# EPICS substitutions: mpgSupport/Db/bsaEdefMaskUnit/bsaEdefMaskUnitAll.substitutions
#==============================================================================
#
# Abs:  Beam Synchronous Acquisition masks
#
# Name: bsaEdefMaskUnitAll.substitutions
#
# Note: Must follow the LCLS naming conventions.
#
#==============================================================================
#
file bsaEdefMaskUnit.db
{
  pattern {     MD,  MASK, INDEX,     SYS ,     DEV   }
	  { $(S_MD), INCM,   1  , $(S_SYS), $(S_DEV)  }
	  { $(S_MD), INCM,   2  , $(S_SYS), $(S_DEV)  }
	  { $(S_MD), INCM,   3  , $(S_SYS), $(S_DEV)  }
          { $(S_MD), INCM,   4  , $(S_SYS), $(S_DEV)  }
          { $(S_MD), INCM,   5  , $(S_SYS), $(S_DEV)  }
          { $(S_MD), INCM,   6  , $(S_SYS), $(S_DEV)  }
          { $(S_MD), INCM,   7  , $(S_SYS), $(S_DEV)  }
          { $(S_MD), INCM,   8  , $(S_SYS), $(S_DEV)  }
          { $(S_MD), INCM,   9  , $(S_SYS), $(S_DEV)  }
          { $(S_MD), INCM,  10  , $(S_SYS), $(S_DEV)  }
          { $(S_MD), INCM,  11  , $(S_SYS), $(S_DEV)  }
          { $(S_MD), INCM,  12  , $(S_SYS), $(S_DEV)  }
          { $(S_MD), INCM,  13  , $(S_SYS), $(S_DEV)  }
          { $(S_MD), INCM,  14  , $(S_SYS), $(S_DEV)  }
          { $(S_MD), INCM,  15  , $(S_SYS), $(S_DEV)  }
          { $(S_MD), INCM,  16  , $(S_SYS), $(S_DEV)  }
          { $(S_MD), INCM,  17  , $(S_SYS), $(S_DEV)  }
          { $(S_MD), INCM,  18  , $(S_SYS), $(S_DEV)  }
          { $(S_MD), INCM,  19  , $(S_SYS), $(S_DEV)  }
          { $(S_MD), INCM,  20  , $(S_SYS), $(S_DEV)  }
          { $(S_MD), INCM,  21  , $(S_SYS), $(S_DEV)  }
          { $(S_MD), INCM,  22  , $(S_SYS), $(S_DEV)  }
          { $(S_MD), INCM,  23  , $(S_SYS), $(S_DEV)  }
          { $(S_MD), INCM,  24  , $(S_SYS), $(S_DEV)  }
          { $(S_MD), INCM,  25  , $(S_SYS), $(S_DEV)  }
          { $(S_MD), INCM,  26  , $(S_SYS), $(S_DEV)  }
          { $(S_MD), INCM,  27  , $(S_SYS), $(S_DEV)  }
          { $(S_MD), INCM,  28  , $(S_SYS), $(S_DEV)  }
          { $(S_MD), INCM,  29  , $(S_SYS), $(S_DEV)  }
          { $(S_MD), INCM,  30  , $(S_SYS), $(S_DEV)  }
          { $(S_MD), INCM,  31  , $(S_SYS), $(S_DEV)  }
          { $(S_MD), INCM,  32  , $(S_SYS), $(S_DEV)  }
          { $(S_MD), INCM,  33  , $(S_SYS), $(S_DEV)  }
          { $(S_MD), INCM,  34  , $(S_SYS), $(S_DEV)  }
          { $(S_MD), INCM,  35  , $(S_SYS), $(S_DEV)  }
          { $(S_MD), INCM,  36  , $(S_SYS), $(S_DEV)  }
          { $(S_MD), INCM,  37  , $(S_SYS), $(S_DEV)  }
          { $(S_MD), INCM,  38  , $(S_SYS), $(S_DEV)  }
          { $(S_MD), INCM,  39  , $(S_SYS), $(S_DEV)  }
          { $(S_MD), INCM,  40  , $(S_SYS), $(S_DEV)  }
          { $(S_MD), INCM,  41  , $(S_SYS), $(S_DEV)  }
          { $(S_MD), INCM,  42  , $(S_SYS), $(S_DEV)  }
          { $(S_MD), INCM,  43  , $(S_SYS), $(S_DEV)  }
          { $(S_MD), INCM,  44  , $(S_SYS), $(S_DEV)  }
          { $(S_MD), INCM,  45  , $(S_SYS), $(S_DEV)  }
          { $(S_MD), INCM,  46  , $(S_SYS), $(S_DEV)  }
          { $(S_MD), INCM,  47  , $(S_SYS), $(S_DEV)  }
          { $(S_MD), INCM,  48  , $(S_SYS), $(S_DEV)  }
          { $(S_MD), INCM,  49  , $(S_SYS), $(S_DEV)  }
          { $(S_MD), INCM,  50  , $(S_SYS), $(S_DEV)  }
          { $(S_MD), INCM,  51  , $(S_SYS), $(S_DEV)  }
          { $(S_MD), INCM,  52  , $(S_SYS), $(S_DEV)  }
          { $(S_MD), INCM,  53  , $(S_SYS), $(S_DEV)  }
          { $(S_MD), INCM,  54  , $(S_SYS), $(S_DEV)  }
          { $(S_MD), INCM,  55  , $(S_SYS), $(S_DEV)  }
          { $(S_MD), INCM,  56  , $(S_SYS), $(S_DEV)  }
          { $(S_MD), INCM,  57  , $(S_SYS), $(S_DEV)  }
          { $(S_MD), INCM,  58  , $(S_SYS), $(S_DEV)  }
          { $(S_MD), INCM,  59  , $(S_SYS), $(S_DEV)  }
          { $(S_MD), INCM,  60  , $(S_SYS), $(S_DEV)  }
          { $(S_MD), INCM,  61  , $(S_SYS), $(S_DEV)  }
          { $(S_MD), INCM,  62  , $(S_SYS), $(S_DEV)  }
          { $(S_MD), INCM,  63  , $(S_SYS), $(S_DEV)  }
          { $(S_MD), INCM,  64  , $(S_SYS), $(S_DEV)  }
          { $(S_MD), INCM,  65  , $(S_SYS), $(S_DEV)  }
          { $(S_MD), INCM,  66  , $(S_SYS), $(S_DEV)  }
          { $(S_MD), INCM,  67  , $(S_SYS), $(S_DEV)  }
          { $(S_MD), INCM,  68  , $(S_SYS), $(S_DEV)  }
          { $(S_MD), INCM,  69  , $(S_SYS), $(S_DEV)  }
          { $(S_MD), INCM,  70  , $(S_SYS), $(S_DEV)  }
          { $(S_MD), INCM,  71  , $(S_SYS), $(S_DEV)  }
          { $(S_MD), INCM,  72  , $(S_SYS), $(S_DEV)  }
          { $(S_MD), INCM,  73  , $(S_SYS), $(S_DEV)  }
          { $(S_MD), INCM,  74  , $(S_SYS), $(S_DEV)  }
          { $(S_MD), INCM,  75  , $(S_SYS), $(S_DEV)  }
          { $(S_MD), INCM,  76  , $(S_SYS), $(S_DEV)  }
          { $(S_MD), INCM,  77  , $(S_SYS), $(S_DEV)  }
          { $(S_MD), INCM,  78  , $(S_SYS), $(S_DEV)  }
          { $(S_MD), INCM,  79  , $(S_SYS), $(S_DEV)  }
          { $(S_MD), INCM,  80  , $(S_SYS), $(S_DEV)  }
          { $(S_MD), INCM,  81  , $(S_SYS), $(S_DEV)  }
          { $(S_MD), INCM,  82  , $(S_SYS), $(S_DEV)  }
          { $(S_MD), INCM,  83  , $(S_SYS), $(S_DEV)  }
          { $(S_MD), INCM,  84  , $(S_SYS), $(S_DEV)  }
          { $(S_MD), INCM,  85  , $(S_SYS), $(S_DEV)  }
          { $(S_MD), INCM,  86  , $(S_SYS), $(S_DEV)  }
          { $(S_MD), INCM,  87  , $(S_SYS), $(S_DEV)  }
          { $(S_MD), INCM,  88  , $(S_SYS), $(S_DEV)  }
          { $(S_MD), INCM,  89  , $(S_SYS), $(S_DEV)  }
          { $(S_MD), INCM,  90  , $(S_SYS), $(S_DEV)  }
          { $(S_MD), INCM,  91  , $(S_SYS), $(S_DEV)  }
          { $(S_MD), INCM,  92  , $(S_SYS), $(S_DEV)  }
          { $(S_MD), INCM,  93  , $(S_SYS), $(S_DEV)  }
          { $(S_MD), INCM,  94  , $(S_SYS), $(S_DEV)  }
          { $(S_MD), INCM,  95  , $(S_SYS), $(S_DEV)  }
          { $(S_MD), INCM,  96  , $(S_SYS), $(S_DEV)  }
          { $(S_MD), INCM,  97  , $(S_SYS), $(S_DEV)  }
          { $(S_MD), INCM,  98  , $(S_SYS), $(S_DEV)  }
          { $(S_MD), INCM,  99  , $(S_SYS), $(S_DEV)  }
          { $(S_MD), INCM, 100  , $(S_SYS), $(S_DEV)  }
          { $(S_MD), INCM, 101  , $(S_SYS), $(S_DEV)  }
          { $(S_MD), INCM, 102  , $(S_SYS), $(S_DEV)  }
          { $(S_MD), INCM, 103  , $(S_SYS), $(S_DEV)  }
          { $(S_MD), INCM, 104  , $(S_SYS), $(S_DEV)  }
          { $(S_MD), INCM, 105  , $(S_SYS), $(S_DEV)  }
          { $(S_MD), INCM, 106  , $(S_SYS), $(S_DEV)  }
          { $(S_MD), INCM, 107  , $(S_SYS), $(S_DEV)  }
          { $(S_MD), INCM, 108  , $(S_SYS), $(S_DEV)  }
          { $(S_MD), INCM, 109  , $(S_SYS), $(S_DEV)  }
          { $(S_MD), INCM, 110  , $(S_SYS), $(S_DEV)  }
          { $(S_MD), INCM, 111  , $(S_SYS), $(S_DEV)  }
          { $(S_MD), INCM, 112  , $(S_SYS), $(S_DEV)  }
          { $(S_MD), INCM, 113  , $(S_SYS), $(S_DEV)  }
          { $(S_MD), INCM, 114  , $(S_SYS), $(S_DEV)  }
          { $(S_MD), INCM, 115  , $(S_SYS), $(S_DEV)  }
          { $(S_MD), INCM, 116  , $(S_SYS), $(S_DEV)  }
          { $(S_MD), INCM, 117  , $(S_SYS), $(S_DEV)  }
          { $(S_MD), INCM, 118  , $(S_SYS), $(S_DEV)  }
          { $(S_MD), INCM, 119  , $(S_SYS), $(S_DEV)  }
          { $(S_MD), INCM, 120  , $(S_SYS), $(S_DEV)  }
          { $(S_MD), INCM, 121  , $(S_SYS), $(S_DEV)  }
          { $(S_MD), INCM, 122  , $(S_SYS), $(S_DEV)  }
          { $(S_MD), INCM, 123  , $(S_SYS), $(S_DEV)  }
          { $(S_MD), INCM, 124  , $(S_SYS), $(S_DEV)  }
          { $(S_MD), INCM, 125  , $(S_SYS), $(S_DEV)  }
          { $(S_MD), INCM, 126  , $(S_SYS), $(S_DEV)  }
          { $(S_MD), INCM, 127  , $(S_SYS), $(S_DEV)  }
          { $(S_MD), INCM, 128  , $(S_SYS), $(S_DEV)  }
          { $(S_MD), INCM, 129  , $(S_SYS), $(S_DEV)  }
          { $(S_MD), INCM, 130  , $(S_SYS), $(S_DEV)  }
          { $(S_MD), INCM, 131  , $(S_SYS), $(S_DEV)  }
          { $(S_MD), INCM, 132  , $(S_SYS), $(S_DEV)  }
          { $(S_MD), INCM, 133  , $(S_SYS), $(S_DEV)  }
          { $(S_MD), INCM, 134  , $(S_SYS), $(S_DEV)  }
          { $(S_MD), INCM, 135  , $(S_SYS), $(S_DEV)  }
          { $(S_MD), INCM, 136  , $(S_SYS), $(S_DEV)  }
          { $(S_MD), INCM, 137  , $(S_SYS), $(S_DEV)  }
          { $(S_MD), INCM, 138  , $(S_SYS), $(S_DEV)  }
          { $(S_MD), INCM, 139  , $(S_SYS), $(S_DEV)  }
          { $(S_MD), INCM, 140  , $(S_SYS), $(S_DEV)  }
          { $(S_MD), INCM, 141  , $(S_SYS), $(S_DEV)  }
          { $(S_MD), INCM, 142  , $(S_SYS), $(S_DEV)  }
          { $(S_MD), INCM, 143  , $(S_SYS), $(S_DEV)  }
          { $(S_MD), INCM, 144  , $(S_SYS), $(S_DEV)  }
          { $(S_MD), INCM, 145  , $(S_SYS), $(S_DEV)  }
          { $(S_MD), INCM, 146  , $(S_SYS), $(S_DEV)  }
          { $(S_MD), INCM, 147  , $(S_SYS), $(S_DEV)  }
          { $(S_MD), INCM, 148  , $(S_SYS), $(S_DEV)  }
          { $(S_MD), INCM, 149  , $(S_SYS), $(S_DEV)  }
          { $(S_MD), INCM, 150  , $(S_SYS), $(S_DEV)  }
          { $(S_MD), INCM, 151  , $(S_SYS), $(S_DEV)  }
          { $(S_MD), INCM, 152  , $(S_SYS), $(S_DEV)  }
          { $(S_MD), INCM, 153  , $(S_SYS), $(S_DEV)  }
          { $(S_MD), INCM, 154  , $(S_SYS), $(S_DEV)  }
          { $(S_MD), INCM, 155  , $(S_SYS), $(S_DEV)  }
          { $(S_MD), INCM, 156  , $(S_SYS), $(S_DEV)  }
          { $(S_MD), INCM, 157  , $(S_SYS), $(S_DEV)  }
          { $(S_MD), INCM, 158  , $(S_SYS), $(S_DEV)  }
          { $(S_MD), INCM, 159  , $(S_SYS), $(S_DEV)  }
          { $(S_MD), INCM, 160  , $(S_SYS), $(S_DEV)  }

	  { $(S_MD), EXCM,   1  , $(S_SYS), $(S_DEV)  }
	  { $(S_MD), EXCM,   2  , $(S_SYS), $(S_DEV)  }
	  { $(S_MD), EXCM,   3  , $(S_SYS), $(S_DEV)  }
          { $(S_MD), EXCM,   4  , $(S_SYS), $(S_DEV)  }
          { $(S_MD), EXCM,   5  , $(S_SYS), $(S_DEV)  }
          { $(S_MD), EXCM,   6  , $(S_SYS), $(S_DEV)  }
          { $(S_MD), EXCM,   7  , $(S_SYS), $(S_DEV)  }
          { $(S_MD), EXCM,   8  , $(S_SYS), $(S_DEV)  }
          { $(S_MD), EXCM,   9  , $(S_SYS), $(S_DEV)  }
          { $(S_MD), EXCM,  10  , $(S_SYS), $(S_DEV)  }
          { $(S_MD), EXCM,  11  , $(S_SYS), $(S_DEV)  }
          { $(S_MD), EXCM,  12  , $(S_SYS), $(S_DEV)  }
          { $(S_MD), EXCM,  13  , $(S_SYS), $(S_DEV)  }
          { $(S_MD), EXCM,  14  , $(S_SYS), $(S_DEV)  }
          { $(S_MD), EXCM,  15  , $(S_SYS), $(S_DEV)  }
          { $(S_MD), EXCM,  16  , $(S_SYS), $(S_DEV)  }
          { $(S_MD), EXCM,  17  , $(S_SYS), $(S_DEV)  }
          { $(S_MD), EXCM,  18  , $(S_SYS), $(S_DEV)  }
          { $(S_MD), EXCM,  19  , $(S_SYS), $(S_DEV)  }
          { $(S_MD), EXCM,  20  , $(S_SYS), $(S_DEV)  }
          { $(S_MD), EXCM,  21  , $(S_SYS), $(S_DEV)  }
          { $(S_MD), EXCM,  22  , $(S_SYS), $(S_DEV)  }
          { $(S_MD), EXCM,  23  , $(S_SYS), $(S_DEV)  }
          { $(S_MD), EXCM,  24  , $(S_SYS), $(S_DEV)  }
          { $(S_MD), EXCM,  25  , $(S_SYS), $(S_DEV)  }
          { $(S_MD), EXCM,  26  , $(S_SYS), $(S_DEV)  }
          { $(S_MD), EXCM,  27  , $(S_SYS), $(S_DEV)  }
          { $(S_MD), EXCM,  28  , $(S_SYS), $(S_DEV)  }
          { $(S_MD), EXCM,  29  , $(S_SYS), $(S_DEV)  }
          { $(S_MD), EXCM,  30  , $(S_SYS), $(S_DEV)  }
          { $(S_MD), EXCM,  31  , $(S_SYS), $(S_DEV)  }
          { $(S_MD), EXCM,  32  , $(S_SYS), $(S_DEV)  }
          { $(S_MD), EXCM,  33  , $(S_SYS), $(S_DEV)  }
          { $(S_MD), EXCM,  34  , $(S_SYS), $(S_DEV)  }
          { $(S_MD), EXCM,  35  , $(S_SYS), $(S_DEV)  }
          { $(S_MD), EXCM,  36  , $(S_SYS), $(S_DEV)  }
          { $(S_MD), EXCM,  37  , $(S_SYS), $(S_DEV)  }
          { $(S_MD), EXCM,  38  , $(S_SYS), $(S_DEV)  }
          { $(S_MD), EXCM,  39  , $(S_SYS), $(S_DEV)  }
          { $(S_MD), EXCM,  40  , $(S_SYS), $(S_DEV)  }
          { $(S_MD), EXCM,  41  , $(S_SYS), $(S_DEV)  }
          { $(S_MD), EXCM,  42  , $(S_SYS), $(S_DEV)  }
          { $(S_MD), EXCM,  43  , $(S_SYS), $(S_DEV)  }
          { $(S_MD), EXCM,  44  , $(S_SYS), $(S_DEV)  }
          { $(S_MD), EXCM,  45  , $(S_SYS), $(S_DEV)  }
          { $(S_MD), EXCM,  46  , $(S_SYS), $(S_DEV)  }
          { $(S_MD), EXCM,  47  , $(S_SYS), $(S_DEV)  }
          { $(S_MD), EXCM,  48  , $(S_SYS), $(S_DEV)  }
          { $(S_MD), EXCM,  49  , $(S_SYS), $(S_DEV)  }
          { $(S_MD), EXCM,  50  , $(S_SYS), $(S_DEV)  }
          { $(S_MD), EXCM,  51  , $(S_SYS), $(S_DEV)  }
          { $(S_MD), EXCM,  52  , $(S_SYS), $(S_DEV)  }
          { $(S_MD), EXCM,  53  , $(S_SYS), $(S_DEV)  }
          { $(S_MD), EXCM,  54  , $(S_SYS), $(S_DEV)  }
          { $(S_MD), EXCM,  55  , $(S_SYS), $(S_DEV)  }
          { $(S_MD), EXCM,  56  , $(S_SYS), $(S_DEV)  }
          { $(S_MD), EXCM,  57  , $(S_SYS), $(S_DEV)  }
          { $(S_MD), EXCM,  58  , $(S_SYS), $(S_DEV)  }
          { $(S_MD), EXCM,  59  , $(S_SYS), $(S_DEV)  }
          { $(S_MD), EXCM,  60  , $(S_SYS), $(S_DEV)  }
          { $(S_MD), EXCM,  61  , $(S_SYS), $(S_DEV)  }
          { $(S_MD), EXCM,  62  , $(S_SYS), $(S_DEV)  }
          { $(S_MD), EXCM,  63  , $(S_SYS), $(S_DEV)  }
          { $(S_MD), EXCM,  64  , $(S_SYS), $(S_DEV)  }
          { $(S_MD), EXCM,  65  , $(S_SYS), $(S_DEV)  }
          { $(S_MD), EXCM,  66  , $(S_SYS), $(S_DEV)  }
          { $(S_MD), EXCM,  67  , $(S_SYS), $(S_DEV)  }
          { $(S_MD), EXCM,  68  , $(S_SYS), $(S_DEV)  }
          { $(S_MD), EXCM,  69  , $(S_SYS), $(S_DEV)  }
          { $(S_MD), EXCM,  70  , $(S_SYS), $(S_DEV)  }
          { $(S_MD), EXCM,  71  , $(S_SYS), $(S_DEV)  }
          { $(S_MD), EXCM,  72  , $(S_SYS), $(S_DEV)  }
          { $(S_MD), EXCM,  73  , $(S_SYS), $(S_DEV)  }
          { $(S_MD), EXCM,  74  , $(S_SYS), $(S_DEV)  }
          { $(S_MD), EXCM,  75  , $(S_SYS), $(S_DEV)  }
          { $(S_MD), EXCM,  76  , $(S_SYS), $(S_DEV)  }
          { $(S_MD), EXCM,  77  , $(S_SYS), $(S_DEV)  }
          { $(S_MD), EXCM,  78  , $(S_SYS), $(S_DEV)  }
          { $(S_MD), EXCM,  79  , $(S_SYS), $(S_DEV)  }
          { $(S_MD), EXCM,  80  , $(S_SYS), $(S_DEV)  }
          { $(S_MD), EXCM,  81  , $(S_SYS), $(S_DEV)  }
          { $(S_MD), EXCM,  82  , $(S_SYS), $(S_DEV)  }
          { $(S_MD), EXCM,  83  , $(S_SYS), $(S_DEV)  }
          { $(S_MD), EXCM,  84  , $(S_SYS), $(S_DEV)  }
          { $(S_MD), EXCM,  85  , $(S_SYS), $(S_DEV)  }
          { $(S_MD), EXCM,  86  , $(S_SYS), $(S_DEV)  }
          { $(S_MD), EXCM,  87  , $(S_SYS), $(S_DEV)  }
          { $(S_MD), EXCM,  88  , $(S_SYS), $(S_DEV)  }
          { $(S_MD), EXCM,  89  , $(S_SYS), $(S_DEV)  }
          { $(S_MD), EXCM,  90  , $(S_SYS), $(S_DEV)  }
          { $(S_MD), EXCM,  91  , $(S_SYS), $(S_DEV)  }
          { $(S_MD), EXCM,  92  , $(S_SYS), $(S_DEV)  }
          { $(S_MD), EXCM,  93  , $(S_SYS), $(S_DEV)  }
          { $(S_MD), EXCM,  94  , $(S_SYS), $(S_DEV)  }
          { $(S_MD), EXCM,  95  , $(S_SYS), $(S_DEV)  }
          { $(S_MD), EXCM,  96  , $(S_SYS), $(S_DEV)  }
          { $(S_MD), EXCM,  97  , $(S_SYS), $(S_DEV)  }
          { $(S_MD), EXCM,  98  , $(S_SYS), $(S_DEV)  }
          { $(S_MD), EXCM,  99  , $(S_SYS), $(S_DEV)  }
          { $(S_MD), EXCM, 100  , $(S_SYS), $(S_DEV)  }
          { $(S_MD), EXCM, 101  , $(S_SYS), $(S_DEV)  }
          { $(S_MD), EXCM, 102  , $(S_SYS), $(S_DEV)  }
          { $(S_MD), EXCM, 103  , $(S_SYS), $(S_DEV)  }
          { $(S_MD), EXCM, 104  , $(S_SYS), $(S_DEV)  }
          { $(S_MD), EXCM, 105  , $(S_SYS), $(S_DEV)  }
          { $(S_MD), EXCM, 106  , $(S_SYS), $(S_DEV)  }
          { $(S_MD), EXCM, 107  , $(S_SYS), $(S_DEV)  }
          { $(S_MD), EXCM, 108  , $(S_SYS), $(S_DEV)  }
          { $(S_MD), EXCM, 109  , $(S_SYS), $(S_DEV)  }
          { $(S_MD), EXCM, 110  , $(S_SYS), $(S_DEV)  }
          { $(S_MD), EXCM, 111  , $(S_SYS), $(S_DEV)  }
          { $(S_MD), EXCM, 112  , $(S_SYS), $(S_DEV)  }
          { $(S_MD), EXCM, 113  , $(S_SYS), $(S_DEV)  }
          { $(S_MD), EXCM, 114  , $(S_SYS), $(S_DEV)  }
          { $(S_MD), EXCM, 115  , $(S_SYS), $(S_DEV)  }
          { $(S_MD), EXCM, 116  , $(S_SYS), $(S_DEV)  }
          { $(S_MD), EXCM, 117  , $(S_SYS), $(S_DEV)  }
          { $(S_MD), EXCM, 118  , $(S_SYS), $(S_DEV)  }
          { $(S_MD), EXCM, 119  , $(S_SYS), $(S_DEV)  }
          { $(S_MD), EXCM, 120  , $(S_SYS), $(S_DEV)  }
          { $(S_MD), EXCM, 121  , $(S_SYS), $(S_DEV)  }
          { $(S_MD), EXCM, 122  , $(S_SYS), $(S_DEV)  }
          { $(S_MD), EXCM, 123  , $(S_SYS), $(S_DEV)  }
          { $(S_MD), EXCM, 124  , $(S_SYS), $(S_DEV)  }
          { $(S_MD), EXCM, 125  , $(S_SYS), $(S_DEV)  }
          { $(S_MD), EXCM, 126  , $(S_SYS), $(S_DEV)  }
          { $(S_MD), EXCM, 127  , $(S_SYS), $(S_DEV)  }
          { $(S_MD), EXCM, 128  , $(S_SYS), $(S_DEV)  }
          { $(S_MD), EXCM, 129  , $(S_SYS), $(S_DEV)  }
          { $(S_MD), EXCM, 130  , $(S_SYS), $(S_DEV)  }
          { $(S_MD), EXCM, 131  , $(S_SYS), $(S_DEV)  }
          { $(S_MD), EXCM, 132  , $(S_SYS), $(S_DEV)  }
          { $(S_MD), EXCM, 133  , $(S_SYS), $(S_DEV)  }
          { $(S_MD), EXCM, 134  , $(S_SYS), $(S_DEV)  }
          { $(S_MD), EXCM, 135  , $(S_SYS), $(S_DEV)  }
          { $(S_MD), EXCM, 136  , $(S_SYS), $(S_DEV)  }
          { $(S_MD), EXCM, 137  , $(S_SYS), $(S_DEV)  }
          { $(S_MD), EXCM, 138  , $(S_SYS), $(S_DEV)  }
          { $(S_MD), EXCM, 139  , $(S_SYS), $(S_DEV)  }
          { $(S_MD), EXCM, 140  , $(S_SYS), $(S_DEV)  }
          { $(S_MD), EXCM, 141  , $(S_SYS), $(S_DEV)  }
          { $(S_MD), EXCM, 142  , $(S_SYS), $(S_DEV)  }
          { $(S_MD), EXCM, 143  , $(S_SYS), $(S_DEV)  }
          { $(S_MD), EXCM, 144  , $(S_SYS), $(S_DEV)  }
          { $(S_MD), EXCM, 145  , $(S_SYS), $(S_DEV)  }
          { $(S_MD), EXCM, 146  , $(S_SYS), $(S_DEV)  }
          { $(S_MD), EXCM, 147  , $(S_SYS), $(S_DEV)  }
          { $(S_MD), EXCM, 148  , $(S_SYS), $(S_DEV)  }
          { $(S_MD), EXCM, 149  , $(S_SYS), $(S_DEV)  }
          { $(S_MD), EXCM, 150  , $(S_SYS), $(S_DEV)  }
          { $(S_MD), EXCM, 151  , $(S_SYS), $(S_DEV)  }
          { $(S_MD), EXCM, 152  , $(S_SYS), $(S_DEV)  }
          { $(S_MD), EXCM, 153  , $(S_SYS), $(S_DEV)  }
          { $(S_MD), EXCM, 154  , $(S_SYS), $(S_DEV)  }
          { $(S_MD), EXCM, 155  , $(S_SYS), $(S_DEV)  }
          { $(S_MD), EXCM, 156  , $(S_SYS), $(S_DEV)  }
          { $(S_MD), EXCM, 157  , $(S_SYS), $(S_DEV)  }
          { $(S_MD), EXCM, 158  , $(S_SYS), $(S_DEV)  }
          { $(S_MD), EXCM, 159  , $(S_SYS), $(S_DEV)  }
          { $(S_MD), EXCM, 160  , $(S_SYS), $(S_DEV)  }
}
